// LS Electric XG5000 project: 16-23-1
// PLC NewPLC
// module base 0 slot 0: 입출력 모듈:XBC-DN/DP14E (DC 24V 입력 8점, 트랜지스터 출력 6점)

PROGRAM NewProgram (task: 스캔 프로그램)

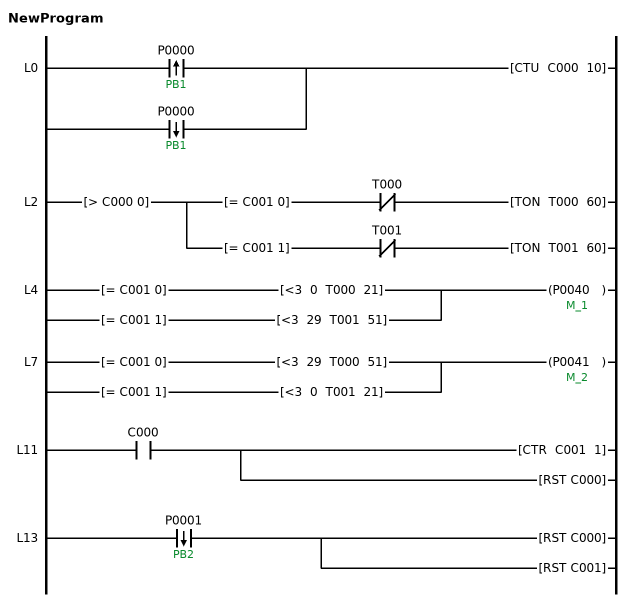
; L0
LOADP     P0000	// PB1
ORN       P0000	// PB1
CTU       C000 10
; L2
LOAD>     C000 0
MPUSH
AND=      C001 0
AND NOT   T000
TON       T000 60
MPOP
AND=      C001 1
AND NOT   T001
TON       T001 60
; L4
LOAD=     C001 0
AND<3     0 T000 21
LOAD=     C001 1
AND<3     29 T001 51
OR LOAD
OUT       P0040	// M_1
; L7
LOAD=     C001 0
AND<3     29 T000 51
LOAD=     C001 1
AND<3     0 T001 21
OR LOAD
OUT       P0041	// M_2
; L11
LOAD      C000
CTR       C001 1
RST       C000
; L13
LOADN     P0001	// PB2
RST       C000
RST       C001